// TIA Portal V16 export
// export: Created 2024-12-03T15:41:45.3481838Z, ExportSetting WithReadOnly, DisplayName Totally Integrated Automation Portal, DisplayVersion V16 Update 6, DisplayName TIA Portal Version Control Interface, DisplayVersion V16 Update 2, DisplayName TIA Portal Openness, DisplayVersion V16 Update 6, DisplayName TIA Portal Teamcenter Gateway, DisplayVersion V16, DisplayName SINAMICS Startdrive Advanced, DisplayVersion V16 Update 5, DisplayName SINAMICS Startdrive G130, G150, S120, S150, SINAMICS MV, S210, DisplayVersion V16 Update 5, DisplayName SINAMICS Startdrive G110M, G120, G120C, G120D, G120P, G115D, DisplayVersion V16 Update 5, DisplayName STEP 7 Professional, DisplayVersion V16 Update 6, DisplayName STEP 7 Safety, DisplayVersion V16, DisplayName WinCC Advanced / Unified PC, DisplayVersion V16 Update 6
TYPE "COGNEX_DATAMAN_OUT_CONTROL_UDT"
// stored: CreationDate 2022-02-10T08:20:21.8932261Z, InterfaceModifiedDate 2022-02-10T08:21:09.6650426Z, IsConsistent true, LibraryConformanceStatus The object is library-conformant., ModifiedDate 2022-02-10T08:21:09.6650426Z
   STRUCT
      ResultBufferEnable : Bool;   // Enables queuing of “Result Data”. If enabled, the current result data will remainuntil acknowledged (even if new results arrive). New results are queued. The nextset of results are pulled from the queue (made available in the Result Datamodule) each time the current results are acknowledged. The DataMan willrespond to the acknowledge by clearing the “Results Available” bit. Once the“Results Ack” bit is cleared the next set of read results will be posted and “ResultsAvailable” will be set True. If results buffering is not enabled newly received readresults will simply overwrite the content of the Result Data module. The reader canbuffer up to 50 and the base station can buffer up to 500 sets of read results
      ResultsAck : Bool;
      spare2 : Bool;
      spare3 : Bool;
      spare4 : Bool;
      spare5 : Bool;
      spare6 : Bool;
      spare7 : Bool;
   END_STRUCT;
END_TYPE
